Universal Robots URScript: vert path wp save.script

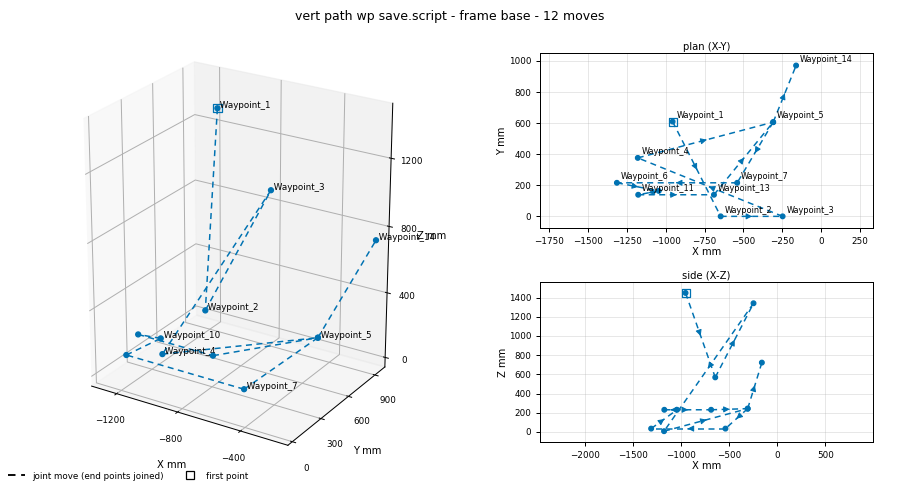
[picture p0: tool path of vert path wp save.script in frame base, 12 of 13 moves have a stored position in this frame; points joined in program order, loops and branches not executed]
def vert_path_wp_save():
  global _hidden_verificationVariable=0
  step_count_ef4628b7_3bf4_4344_8274_e41c2c4e5143 = 0.0
  thread Step_Counter_Thread_73ad19e4_304f_4293_8782_e512d608e2cc():
    while (True):
      step_count_ef4628b7_3bf4_4344_8274_e41c2c4e5143 = step_count_ef4628b7_3bf4_4344_8274_e41c2c4e5143 + 1.0
      sync()
    end
  end
  run Step_Counter_Thread_73ad19e4_304f_4293_8782_e512d608e2cc()
  set_safety_mode_transition_hardness(1)
  set_tool_communication(False, 115200, 0, 1, 1.5, 3.5)
  set_tool_output_mode(0)
  set_tool_digital_output_mode(0, 1)
  set_tool_digital_output_mode(1, 1)
  set_tool_voltage(0)
  set_tcp(p[-0.0042110779091591305,-0.2798289119592719,0.10591607363377763,1.2092,-1.2092,1.2092])
  set_standard_analog_input_domain(0, 1)
  set_standard_analog_input_domain(1, 1)
  set_tool_analog_input_domain(0, 1)
  set_tool_analog_input_domain(1, 1)
  set_analog_outputdomain(0, 0)
  set_analog_outputdomain(1, 0)
  set_input_actions_to_default()
  set_gravity([0.0, 0.0, 9.82])
  set_target_payload(7.750000, [0.000000, -0.007000, 0.070000], [0.046720, 0.046720, 0.046720, 0.000000, 0.000000, 0.000000])
  global Point_1=p[0.0,0.0,0.0,0.0,0.0,0.0]
  # begin: URCap Installation Node
  #   Source: MachineLogic for Universal Robots, 3.1.7, Vention Inc.
  #   Type: MachineLogic for Universal Robots
  def waitForResponse(expected_response_vention, cname_vention):
  response_vention = socket_read_string(cname_vention,timeout=15)
  while response_vention != expected_response_vention:
  sleep(0.01)
  response_vention = socket_read_string(cname_vention,timeout=15)
  end
  sleep(0.01)
  sync()
  end
  def sendString(string_vention, expected_response_vention, cname_vention):
  socket_send_string(str_cat(string_vention,";"), cname_vention)
  response_vention = socket_read_string(cname_vention,timeout=15)
  if(response_vention == "nAck"):
  popup("nAck received")
  end
  while response_vention != expected_response_vention:
  sleep(0.01)
  response_vention = socket_read_string(cname_vention,timeout=15)
  if(response_vention == "nAck"):
  popup("nAck received")
  end
  end
  sleep(0.01)
  sync()
  end
  def sendStringNAck(string_vention, expected_response_vention, cname_vention):
  socket_send_string(str_cat(string_vention,";"), cname_vention)
  response_vention = socket_read_string(cname_vention,timeout=15)
  if(response_vention == "nAck"):
  popup("nAck received")
  end
  while(response_vention != expected_response_vention and response_vention != "nAck"):
  sleep(0.01)
  response_vention = socket_read_string(cname_vention,timeout=15)
  if(response_vention == "nAck"):
  popup("nAck received",blocking=True)
  end
  end
  sleep(0.01)
  sync()
  end
  def sendStringWithTimeout(string_vention, expected_response_vention, cname_vention):
  socket_send_string(str_cat(string_vention,";"), cname_vention)
  response_vention = socket_read_string(cname_vention,timeout=10)
  if(response_vention == "nAck"):
  popup("nAck received"+string_vention)
  end
  sleep(0.01)
  sync()
  end
  def pollString(string_vention, expected_response_vention, cname_vention):
  socket_send_string(str_cat(string_vention,";"), cname_vention)
  response_vention = socket_read_string(cname_vention,timeout=15)
  if(response_vention == "nAck"):
  popup("nAck received")
  end
  while response_vention != expected_response_vention:
  sleep(1)
  socket_send_string(str_cat(string_vention,";"), cname_vention)
  response_vention = socket_read_string(cname_vention,timeout=15)
  if(response_vention == "nAck"):
  popup("nAck received")
  end
  end
  sleep(0.01)
  sync()
  end
  def sendVariable(var_vention, data_vention, expected_response_vention, cname_vention):
  socket_set_var(var_vention, data_vention, cname_vention)
  response_vention = socket_read_string(cname_vention,timeout=15)
  if(response_vention == "nAck"):
  popup("nAck received")
  end
  while response_vention != expected_response_vention:
  sleep(0.01)
  response_vention = socket_read_string(cname_vention,timeout=15)
  if(response_vention == "nAck"):
  popup("nAck received")
  end
  end
  sleep(0.01)
  sync()
  end
  def intToString(integer_vention,cname_vention):
  stringFix=""
  multiplier_vention123=1
  if integer_vention<0:
  stringFix="-"
  multiplier_vention123=-1
  end
  socket_set_var("GetString",integer_vention*multiplier_vention123,cname_vention)
  string_vention=""
  while string_vention=="":
  sleep(0.01)
  string_vention=socket_read_string(cname_vention,timeout=15)
  end
  sleep(0.01)
  sync()
  string_vention=stringFix+string_vention
  return string_vention
  end
  string_vention=""
  isVentionMovementBusy = False
  isVentionParallelMovementSendingScript = False
  ventionThreadHandle = 1
  isVentionMovementBusyMachineMotion1 = False
  isVentionParallelMovementSendingScriptMachineMotion1 = False
  socket_vention = socket_open("192.168.3.52", 9999, "MachineMotion1")
  if socket_vention==False:
  popup("Check configuration, can't connect to MachineMotion")
  end
  waitForResponse("MachineMotion connection established", "MachineMotion1")
  sendString("isReady", "MachineMotion isReady = true", "MachineMotion1")
  sendStringWithTimeout("setURCapVersion2", "setURCapVersion loaded", "MachineMotion1")
  sendString("SET speed_v2 1000000", "Ack", "MachineMotion1")
  sendString("SET acceleration_v2 100000", "Ack", "MachineMotion1")
  sendString("SET de_axis_1_microsteps_config 8", "Ack", "MachineMotion1")
  sendString("SET de_axis_1_mechanical_gain_config_v2 150000.0", "Ack", "MachineMotion1")
  sendString("SET de_axis_1_direction_config 1", "Ack", "MachineMotion1")
  sendString("SET de_axis_1_type_config Custom Actuator ", "Ack", "MachineMotion1")
  sendString("de_axis_1_config_exec", "Ack", "MachineMotion1")
  # end: URCap Installation Node
  global Waypoint_1_p=p[-.955652198299, .609645262545, 1.447606621703, -.000002586602, .000023983690, -.000044728674]
  global Waypoint_1_q=[-0.6190655867206019, -0.3368618053248902, -0.41324496269226074, 3.89075676977124, 2.190887689590454, -4.6617189516240387E-4]
  global Waypoint_2_p=p[-.646472006716, -.000005175669, .568192325689, -.000000485067, -.000006973981, -.000005045961]
  global Waypoint_2_q=[-0.23332149187196904, 0.9707986551472167, -1.9700188636779785, 4.139979048366211, 1.8039493560791016, -2.5588670839482575E-4]
  global Waypoint_3_p=p[-.247841618163, -.000001221844, 1.340099232237, 1.570793608201, -.000028410849, -.000016022498]
  global Waypoint_3_q=[-0.8519218603717249, -0.33198924482379155, -1.6308417320251465, 5.1035817740257166, 2.42344331741333, 1.5703715085983276]
  global Waypoint_4_p=p[-1.179747427322, .376142202196, .007542577009, 1.379988252251, -.891987002417, -.892019582121]
  global Waypoint_4_q=[-0.7655184904681605, -0.2574165624431153, 1.2221644560443323, 2.1762491899677734, 1.189542293548584, 1.5704518556594849]
  global Waypoint_5_p=p[-.308518516300, .606106971306, .242383883754, -2.133736308583, .349453533645, 2.130945814092]
  global Waypoint_5_q=[-1.8566301504718226, -1.2938345235637208, 2.2087047735797327, 0.7414883810230712, 1.586585521697998, 1.5234099626541138]
  global Waypoint_7_p=p[-.540145657443, .215928159451, .034626615128, -1.505818452622, 1.057589549975, 1.573496338188]
  global Waypoint_7_q=[-0.4478219191180628, -1.1245789390853425, 2.485603157673971, 0.16253535329785151, 1.4958982467651367, 3.833399772644043]
  global Waypoint_6_p=p[-1.314145372626, .215925160668, .034627130433, -1.505810875646, 1.057606245516, 1.573489538167]
  global Waypoint_6_q=[-0.14954883257021123, -0.5748068255237122, 1.1567109266864222, 0.9217995840260009, 1.512316107749939, 4.131750583648682]
  global Waypoint_10_p=p[-1.044592918419, .163806109417, .230713077830, -.897773218539, -1.600868829001, 1.600908850228]
  global Waypoint_10_q=[-0.4298151175128382, -1.2030299764922638, 2.2937288920031946, 5.192346173315801, -4.1211939493762415, 1.571419358253479]
  global Waypoint_11_p=p[-1.176999957936, .138945371956, .230679149733, -.852011383486, -1.646009308825, 1.646012828723]
  global Waypoint_11_q=[-0.3604524771319788, -1.107452170257904, 2.1078084150897425, 5.282046007900991, -4.11819297472109, 1.5714211463928223]
  global Waypoint_13_p=p[-.689653194730, .138979794491, .230695810576, -.851995676063, -1.645986640376, 1.645983874930]
  global Waypoint_13_q=[-0.9414122740374964, -1.5014984545162697, 2.8018503824817103, 4.981593298702993, -4.698930088673727, 1.5716490745544434]
  global Waypoint_12_p=p[-.308525731278, .606094712829, .242387732524, 1.369874344706, 1.066885302939, -1.257203969235]
  global Waypoint_12_q=[-1.4685633818255823, -0.9664476078799744, 1.6195014158831995, 0.9282733637043457, 1.6574419736862183, 0.2630743682384491]
  global Waypoint_14_p=p[-.161041255041, .970521625376, .722022711392, -.554981128664, .106460999224, .328583716452]
  global Waypoint_14_q=[-1.3071578184710901, -1.3366714429906388, 2.2083800474749964, 3.7187773424335937, -2.9519384543048304, 0.9132328033447266]
  while (True):
    $ 2 "Robot Program"
    $ 3 "Home"
    movej([-3.523764549353853, -1.8742328384451357, 2.4457816539194326, 0.058650484450722296, -0.22275931369636837, -0.6273979632655688], a=1.3962634015954636, v=1.0471975511965976)
    $ 4 "MoveJ"
    $ 5 "Waypoint_1" "breakAfter"
    movej(get_inverse_kin(Waypoint_1_p, qnear=Waypoint_1_q), t=2.0)
    $ 6 "Waypoint_2" "breakAfter"
    movej(get_inverse_kin(Waypoint_2_p, qnear=Waypoint_2_q), a=1.3962634015954636, v=1.0471975511965976)
    $ 7 "Waypoint_3" "breakAfter"
    movej(get_inverse_kin(Waypoint_3_p, qnear=Waypoint_3_q), a=1.3962634015954636, v=1.0471975511965976)
    $ 8 "MoveJ"
    $ 9 "Waypoint_4" "breakAfter"
    movej(get_inverse_kin(Waypoint_4_p, qnear=Waypoint_4_q), a=1.3962634015954636, v=1.0471975511965976)
    $ 10 "Waypoint_5" "breakAfter"
    movej(get_inverse_kin(Waypoint_5_p, qnear=Waypoint_5_q), a=1.3962634015954636, v=1.0471975511965976)
    $ 11 "Waypoint_7" "breakAfter"
    movej(get_inverse_kin(Waypoint_7_p, qnear=Waypoint_7_q), a=1.3962634015954636, v=1.0471975511965976)
    $ 12 "Waypoint_6" "breakAfter"
    movej(get_inverse_kin(Waypoint_6_p, qnear=Waypoint_6_q), a=1.3962634015954636, v=1.0471975511965976)
    $ 13 "'the waypoints for getting from home to DOtA down'"
    # 'the waypoints for getting from home to DOtA down'
    $ 14 "MoveJ"
    $ 17 "Waypoint_10" "breakAfter"
    movej(get_inverse_kin(Waypoint_10_p, qnear=Waypoint_10_q), a=1.3962634015954636, v=1.0471975511965976)
    $ 18 "Waypoint_11" "breakAfter"
    movej(get_inverse_kin(Waypoint_11_p, qnear=Waypoint_11_q), a=1.3962634015954636, v=1.0471975511965976)
    $ 19 "Waypoint_13" "breakAfter"
    movej(get_inverse_kin(Waypoint_13_p, qnear=Waypoint_13_q), a=1.3962634015954636, v=1.0471975511965976)
    $ 20 "MoveJ"
    $ 21 "Waypoint_12" "breakAfter"
    movej(get_inverse_kin(Waypoint_12_p, qnear=Waypoint_12_q), a=1.3962634015954636, v=1.0471975511965976)
    $ 22 "Waypoint_14" "breakAfter"
    movej(get_inverse_kin(Waypoint_14_p, qnear=Waypoint_14_q), a=1.3962634015954636, v=1.0471975511965976)
  end
end
